# B&R Automation Studio project BR_SHA256
Automation Studio 4.12.5.95

## Configuration Config1

### Task classes (Cpu.sw)
```
Cyclic#1 (cycle 100 us, tolerance 100 us):
  Program <- (binary)
Cyclic#6:
  BlinkerC <- BlinkerC.prg
  BlinkerL <- BlinkerL.prg
Cyclic#7:
  CycleTime <- CycleTime.prg
  SHA256 <- SHA256.prg
Binaries: udbdef, FWRules, TCData, iomap, ashwac, Role, sysconf, arconfig, asfw, User, ashwd
Libraries: runtime, astime, asieccon
```

### Hardware
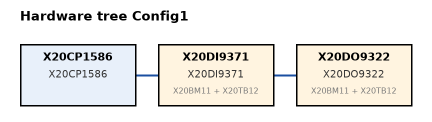
```
X20BM11 : X20BM11 v1.1.0.0  [X2X1 -> X20CP1586.IF6]
X20BM11a : X20BM11 v1.1.0.0  [X2X1 -> X20BM11.X2X2]
X20CP1586 : X20CP1586 v1.10.0.0
  Connector IF2:
    ActivateDevice = 1
  ConfigurationID = X20CP1586AS4_Config1
  Simulation = 1
  SystemTick = 100
  IdleTaskClass = 8
  TaskClassIdleTime = 2000
  Cyclic1Duration = 100
  Cyclic1Tolerance = 100
  Cyclic2Duration = 1000
  Cyclic2Tolerance = 1000
  Cyclic3Duration = 10000
  Cyclic3Tolerance = 10000
  FileDevice1
  FileDeviceName1 = USER
  FileDevicePath1 = USER_PATH
  ActivateSntp = 1
  SntpcServAddr1 = time.google.com
  SntpcServAddr2 = time.aws.com
  SntpcServAddr3 = time.cloudflare.com
  SntpcServAddr4 = time.windows.com
  ActivateOpcUa = 1
  OpcUa_AuthenticationSecurityPolicy_EnableNone = 1
  OpcUa_AuthenticationSecurityPolicy_EnableBasic128Rsa15 = 1
  OpcUaInformationModels_PV_Version = 1
X20DI9371 : X20DI9371 v1.4.0.0  [SS1 -> X20TB12.SS; SL -> X20BM11.SL1]
X20DO9322 : X20DO9322 v1.5.0.0  [SS1 -> X20TB12a.SS; SL -> X20BM11a.SL1]
X20TB12 : X20TB12 v1.0.0.0
X20TB12a : X20TB12 v1.0.0.0
```

## Logical view

### Program Logical/CycleTime

#### Variables.var
```iecst
VAR
	CycleTimeTicks : LREAL;
END_VAR
```

#### Main.c
```c
#include <bur/plctypes.h>
#include <inttypes.h>

#ifdef _DEFAULT_INCLUDES
	#include <AsDefault.h>
#endif

static uint64_t cycles, cycles_saved;

uint64_t rdtsc() {
	uint32_t low, high;
	__asm__ __volatile__(
		"rdtsc"
		: "=a" (low),
		"=d" (high)
	);
	return ((uint64_t)high << 32) | low;
}

void _INIT ProgramInit(void)
{
	cycles_saved = rdtsc();

}

void _CYCLIC ProgramCyclic(void)
{
	cycles = rdtsc();
	CycleTimeTicks = (LREAL)(cycles - cycles_saved);
	cycles_saved = cycles;
}

void _EXIT ProgramExit(void)
{

}
```

### Program Logical/SHA256

#### Main.c
```c
#include <bur/plctypes.h>

#ifdef _DEFAULT_INCLUDES
#include <AsDefault.h>
#endif

#include "sha256.h"

static long long begin, begin_saved, end;

long long rdtsc() {
	unsigned int low, high;
	__asm__ __volatile__("rdtsc" : "=a" (low), "=d" (high));
		return ((long long)high << 32) | low;
}

void _INIT ProgramInit(void)
{
	int i; //C99
	for(i = 0; i< sizeof(buffer); i++) buffer[i] = 'a';
	cycles_counter = 0;
}

void _CYCLIC ProgramCyclic(void)
{
	SHA256_CTX ctx;

	begin = rdtsc();
	cycle_time = (LREAL)(begin - begin_saved);
	begin_saved = begin;

	sha256_init(&ctx);
	sha256_update(&ctx, buffer, sizeof(buffer));
	sha256_final(&ctx, digest);

	end = rdtsc();
	cpu_time_used = ((LREAL)(end - begin));

	MBperSec = cycle_time / cpu_time_used;
	cycles_counter++;
}

void _EXIT ProgramExit(void) {}
```
